(* PLC project Unnamed, Unknown Unnamed 1 *)
(* stored: creationDateTime 2024-09-14T19:27:39, modificationDateTime 2024-09-15T10:56:18 *)

PROGRAM counter
  VAR
    input_register AT %IW0.0 : INT;
    output_register AT %QW0.0 : INT;
  END_VAR

            (*Needed a basic program to check basic functions of python modbus simulation.*)
(*With this program I was able to change the input register and read the change in the output register.*)
output_register := input_register;
          
END_PROGRAM

CONFIGURATION Config0
  RESOURCE Res0 ON PLC
    TASK task0(INTERVAL := T#20ms, PRIORITY := 0);
    PROGRAM instance0 WITH task0 : counter;
  END_RESOURCE
END_CONFIGURATION
